///////////
// Structure For I35. Main Operating Data to be saved (ex: OPC).  
//////////
TYPE PM_ION9200 :
STRUCT
		MesData						: PM ; (* Object *) 
		MesSeconds					: REAL;
		
		
END_STRUCT
END_TYPE

(* stored: Version 1.1.0.1, ProductVersion 3.1.4024.9
   DUT PM_ION9200: Id {89465405-5c3e-4d53-8bc7-b2a79c03b846} *)
